# EPICS substitutions: rogueApp/Db/AxiVersion.substitutions
# AxiVersion.substitutions

#file biDevRogue.template
#{
#}
file boDevRogue.template
{
	{
		NAME	= "AxiVersion:FpgaReload",
		PATH	= "Top.AxiVersion.FpgaReload",
		PYPV	= "Top:AxiVersion:FpgaReload",
		DESC	= "AxiPcieCore FPGA Reload"
		ZNAM	= "Normal"
		ONAM	= "Reload"
		SAVE	= ""
	}
}
#file boolDevRogue.template
#{
#}

file liDevRogue.template
{
	{
		NAME	= "AxiVersion:FpgaVersion",
		PATH	= "Top.AxiVersion.FpgaVersion",
		PYPV	= "Top:AxiVersion:FpgaVersion",
		DESC	= "AxiPcieCore FPGA Version (show as hex)"
		PINI	= "YES"
	}
	{
		NAME	= "AxiVersion:UpTime",
		PATH	= "Top.AxiVersion.UpTimeCnt",
		PYPV	= "Top:AxiVersion:UpTimeCnt",
		EGU		= "sec"
		SCAN	= "\$(SCAN=1 second)"
	}
}

#file loDevRogue.template
#{
#}

file longDevRogue.template
{
	{
		NAME	= "AxiVersion:ScratchPad",
		PATH	= "Top.AxiVersion.ScratchPad"
		PYPV	= "Top:AxiVersion:ScratchPad"
		PINI	= "YES"
		SAVE	= ""
	}
	{
		NAME	= "AxiVersion:UserReset",
		PATH	= "Top.AxiVersion.UserReset"
		PYPV	= "Top:AxiVersion:UserReset"
		SAVE	= ""
	}
}

#       DESC    = "0         1         2         3         "
#       DESC    = "01234567890123 Max 40 char 7890123456789"
